(* PLC project Tc2_MC2.stLibVersion_Tc2_MC2 Demo, tc3-libraries-kb TwinCAT 3.1 *)
(* stored: creationDateTime 2026-05-21T00:00:00, modificationDateTime 2026-05-21T00:00:00 *)

PROGRAM P_Demo_stLibVersion_Tc2_MC2
  VAR
    bMC2VersionOK : BOOL;  (* 比对结果：≥2.17.0 即 TRUE *)
    sCurrentVersion : STRING;
  END_VAR

// =============================================================================
// 场景：开机自检 — 验证当前链接的 Tc2_MC2 库 ≥ 2.17.0 才允许后续运动使能
// 价值：一行代码避免"现场库版本错乱"导致的隐式行为差异
// 验证：登录后看 bMC2VersionOK 是否 TRUE；sCurrentVersion 是否显示 "2.17.0"
// =============================================================================

// F_CmpLibVersion 在 Tc2_System 库；编译期注入常量，运行时 O(1)
bMC2VersionOK := F_CmpLibVersion(stLibVersion_Tc2_MC2, 2, 17, 0, '>=');
sCurrentVersion := stLibVersion_Tc2_MC2.sVersion;
END_PROGRAM
